{attribute 'qualified_only'}
{attribute 'strict'}
TYPE E_TestStates :
(
    eInitialiseTest := 0,
    ePreparePreTestConditions := 1,
    eExecutePreTestConditions := 2,
    ePrepareTest := 3,
    eExecuteTest := 4,
    eWaitForResults := 5,
    ePrepareFinishTest := 6,
    eExecuteFinishTest := 7,
    eReportFinishedTest := 8
);
END_TYPE

(* stored: Version 1.1.0.1, ProductVersion 3.1.4024.5
   DUT E_TestStates: Id {fa5c3f3c-c558-44f1-8e4d-ea57c6a7bb8e} *)
